// SIMATIC S7-200 project (STEP 7-Micro/WIN), CPU 222 REL 02.01

SYMBOL_TABLE USUARIO1
PARO             I0.0
MARCHA_1         I0.1
MARCHA_2         I0.2
LAMPARA_1        Q0.0
LAMPARA_2        Q0.1
END_SYMBOL_TABLE

ORGANIZATION_BLOCK PRINCIPAL:OB1
TITLE=COMENTARIOS DEL PROGRAMA
BEGIN
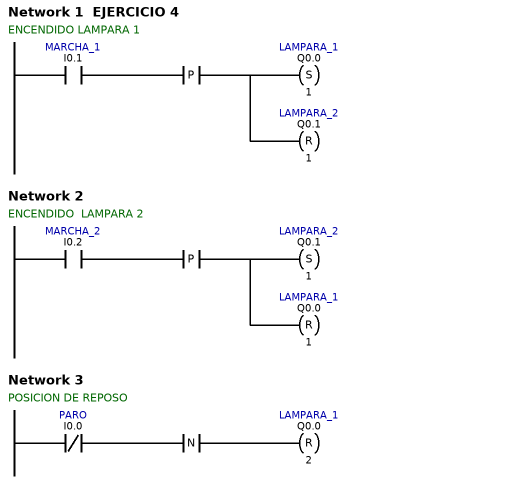
Network 1 // EJERCICIO 4
// ENCENDIDO LAMPARA 1
LD     MARCHA_1:I0.1
EU
S      LAMPARA_1:Q0.0, 1
R      LAMPARA_2:Q0.1, 1
Network 2
// ENCENDIDO  LAMPARA 2 
LD     MARCHA_2:I0.2
EU
S      LAMPARA_2:Q0.1, 1
R      LAMPARA_1:Q0.0, 1
Network 3
// POSICION DE REPOSO 
// (network saved uncompiled; LAD cells follow)
// row 0: c0 -|/|- PARO:I0.0  c1 -|N|-  c2 -(R) LAMPARA_1:Q0.0, 2
END_ORGANIZATION_BLOCK
